TYPE _ST_SiftMessage :
STRUCT
	nType : BYTE;
	nLength : UDINT;
	aData : ARRAY[1..SiftClientParameters.MAX_DATA_MESSAGE_SIZE] OF BYTE;
END_STRUCT
END_TYPE

(* stored: Version 1.1.0.1
   DUT _ST_SiftMessage: Id {3cb988cd-a91a-4ab6-8487-5bc9f1f1555c} *)
